// TwinCAT 3 PLC project step_motor
// ProgramVersion: 3.1.4023.0
// libraries:
//   Tc2_MC2, * (Beckhoff Automation GmbH)
//   Tc2_Standard, * (Beckhoff Automation GmbH)
//   Tc2_System, * (Beckhoff Automation GmbH)
//   Tc3_Module, * (Beckhoff Automation GmbH)
//   VisuSymbols,3.5.10.0,System
// project tree:
//   DUTs/ ST_MC_Status.TcDUT
//   / GlobalTextList.TcGTLO, PlcTask.TcTTO, Visualization Manager.TcVMO (not stored)
//   GVLs/ GVL.TcGVL
//   POUs/ MAIN.TcPOU
//   VISUs/ Visualization.TcVIS
// real-time tasks:
//   TASK PlcTask: cycle T#10ms, priority 20, ADS port 350
// motion (NC):
//   TASK NC-Task 1 SAF: cycle T#2ms, priority 4, ADS port 501
//   TASK NC-Task 1 SVB: cycle T#10ms, priority 8, ADS port 511
//   AXIS Axis 1 (id 1)
//     PositionAreaControl: Enable=false
//     TargetPosControl: Enable=false
//     OtherSettings: AllowMotionCmdToSlave=true
//     encoder EncType=4
//       EncPara: MaxCount=#x0000ffff
//         FilterTime: TPos=0.04, TVelo=0.1, TAcc=0.15
//         Inc: RefMode=2, RefSoftSyncMask=#x0000ffff
//     drive DrvType=24
//       Analog: VeloReferenz=800, TorqueSetpointScale=10, ScaleFactorActTorque=0.1
//       TimeComp: TaskDelayCycles=1
//     controller CtrType=1
//       CtrPara: PriorControlFactor=1
//         PosDiffControl: Enable=false
//         Observer: BandWidth=20
// I/O:
//   DEVICE Device 1 (EtherCAT), AmsNetId 5.59.220.46.2.1
//     Term 7 (EK1200) [EK1200-5000 EtherCAT Power supply (2A E-Bus)]
//       Term 8 (EL1008) [EL1008 8Ch. Dig. Input 24V, 3ms]
//       Term 9 (EL2008) [EL2008 8Ch. Dig. Output 24V, 0.5A]
//       Term 10 (EL3062) [EL3062 2Ch. Ana. Input 0-10V]
//       Term 11 (EL4002) [EL4002 2Ch. Ana. Output 0-10V, 12bit]
//       Term 12 (EL7031) [EL7031 1Ch. Stepper motor output stage (24V, 1.5A)]
//       Term 13 (EK1110) [EK1110 EtherCAT extension]
// variable links:
//   NC-Task 1 SAF/Axes/Axis 1 <-> Device 1 (EtherCAT)/Term 7 (EK1200)/Term 12 (EL7031)
//     Drive/Inputs/In/nState1 @bit 3 <-> STM Status/Status/Error
//     Drive/Inputs/In/nState1 @bit 5 <-> STM Status/Status/Moving negative
//     Drive/Inputs/In/nState1 @bit 4 <-> STM Status/Status/Moving positive
//     Drive/Inputs/In/nState1 @bit 1 <-> STM Status/Status/Ready
//     Drive/Inputs/In/nState1 <-> STM Status/Status/Ready to enable
//     Drive/Inputs/In/nState1 @bit 6 <-> STM Status/Status/Torque reduced
//     Drive/Inputs/In/nState1 @bit 2 <-> STM Status/Status/Warning
//     Drive/Inputs/In/nState2 @bit 3 <-> STM Status/Status/Digital input 1
//     Drive/Inputs/In/nState2 @bit 4 <-> STM Status/Status/Digital input 2
//     Drive/Inputs/In/nState2 @bit 5 <-> STM Status/Status/Sync error
//     Drive/Inputs/In/nState2 @bit 7 <-> STM Status/Status/TxPDO Toggle
//     Drive/Inputs/In/nState4 @bit 1 <-> WcState/InputToggle
//     Drive/Inputs/In/nState4 <-> WcState/WcState
//     Drive/Outputs/Out/nCtrl1 <-> STM Control/Control/Enable
//     Drive/Outputs/Out/nCtrl1 @bit 2 <-> STM Control/Control/Reduce torque
//     Drive/Outputs/Out/nCtrl1 @bit 1 <-> STM Control/Control/Reset
//     Drive/Outputs/Out/nDataOut2[0] <-> STM Velocity/Velocity
//     Enc/Inputs/In/nDataIn1[0] <-> ENC Status compact/Counter value
//     Enc/Inputs/In/nDataIn2[0] <-> ENC Status compact/Latch value
//     Enc/Inputs/In/nState1 @bit 4 <-> ENC Status compact/Status/Counter overflow
//     Enc/Inputs/In/nState1 @bit 3 <-> ENC Status compact/Status/Counter underflow
//     Enc/Inputs/In/nState1 @bit 1 <-> ENC Status compact/Status/Latch extern valid
//     Enc/Inputs/In/nState1 @bit 2 <-> ENC Status compact/Status/Set counter done
//     Enc/Inputs/In/nState2 @bit 4 <-> ENC Status compact/Status/Status of extern latch
//     Enc/Inputs/In/nState2 @bit 5 <-> ENC Status compact/Status/Sync error
//     Enc/Inputs/In/nState2 @bit 7 <-> ENC Status compact/Status/TxPDO Toggle
//     Enc/Inputs/In/nState4 @bit 1 <-> WcState/InputToggle
//     Enc/Inputs/In/nState4 <-> WcState/WcState
//     Enc/Outputs/Out/nCtrl1 @bit 3 <-> ENC Control compact/Control/Enable latch extern on negative edge
//     Enc/Outputs/Out/nCtrl1 @bit 1 <-> ENC Control compact/Control/Enable latch extern on positive edge
//     Enc/Outputs/Out/nCtrl1 @bit 2 <-> ENC Control compact/Control/Set counter
//     Enc/Outputs/Out/nDataOut1[0] <-> ENC Control compact/Set counter value
//   step_motor/step_motor Instance <-> NC-Task 1 SAF/Axes/Axis 1
//     PlcTask Inputs/MAIN.Axis.NcToPlc <-> Outputs/ToPlc
//     PlcTask Outputs/MAIN.Axis.PlcToNc <-> Inputs/FromPlc

CONFIGURATION step_motor
    RESOURCE PLC ON TwinCAT3
        TASK PlcTask(INTERVAL := T#10ms, PRIORITY := 20);
        PROGRAM MAIN WITH PlcTask : MAIN;
    END_RESOURCE
END_CONFIGURATION

// ---- DUTs/ST_MC_Status.TcDUT
TYPE ST_MC_Status :
STRUCT
	Status 		: BOOL;
	Done   		: BOOL;
	Busy   		: BOOL;
	Error  		: BOOL;
	Active 		: BOOL;
	CadAborted	: BOOL;
	InVelocity	: BOOL;
	ErrorID		: UDINT;
END_STRUCT
END_TYPE

// ---- GVLs/GVL.TcGVL
{attribute 'qualified_only'}
VAR_GLOBAL
	// Axis
	Axis: AXIS_REF;
	
	// Function blocks
	fbPowerAxis: MC_Power;
	fbMoveContinuous: MC_MoveContinuousRelative;
	
	// Parameters
	
	PowerOverride	: LREAL := 100;
	
	// Status
	
	Power 		  : ST_MC_Status;
	MoveRelative  : ST_MC_Status;
	Jog			  : ST_MC_Status;
END_VAR

// ---- POUs/MAIN.TcPOU
PROGRAM MAIN
VAR
	fbPowerAxis: MC_Power;
	fbMoveContinuous  : MC_MoveContinuousRelative;
	MC_Jog : MC_Jog;
		
	Axis: AXIS_REF;
	bExecute, bEnable: BOOL;
    bEnableP, bEnableN: BOOL := TRUE;
	rVelocity : LREAL := 600;
	rDistance : LREAL := 360;
END_VAR

GVL.fbPowerAxis(
	Axis:= GVL.Axis,
	Enable:= bEnable, 
	Enable_Positive:= bEnableP, 
	Enable_Negative:= bEnableN, 
	Override:= GVL.PowerOverride, 
	BufferMode:= MC_Aborting, 
	Options:= , 
	Status=> GVL.Power.Status, 
	Busy=> GVL.Power.Busy, 
	Active=> GVL.Power.Active, 
	Error=> GVL.Power.Error, 
	ErrorID=> gvl.Power.ErrorID);
	
	
(*GVL.fbMoveContinuous(
	Axis:= GVL.Axis, 
	Execute:= bExecute, 
	Distance:= rDistance, 
	Velocity:= rVelocity, 
	EndVelocity:= rVelocity, 
	Acceleration:= 500, 
	Deceleration:= 500, 
	Jerk:= 10, 
	BufferMode:= MC_Aborting, 
	Options:= , 
	InEndVelocity=> GVL.MoveRelative.InVelocity, 
	Busy=> GVL.MoveRelative.Busy, 
	Active=> GVL.MoveRelative.Active, 
	CommandAborted=> GVL.MoveRelative.CadAborted, 
	Error=> GVL.MoveRelative.Error, 
	ErrorID=> GVL.MoveRelative.ErrorID);*)
	
	(*MC_Jog(
	Axis:= GVL.Axis, 
	JogForward:= , 
	JogBackwards:= , 
	Mode:= MC_JOGMODE_CONTINOUS, 
	Position:= rDistance, 
	Velocity:= rVelocity, 
	Acceleration:= 500, 
	Deceleration:= 500, 
	Jerk:= 10, 
	Done=> GVL.Jog.Done, 
	Busy=> GVL.Jog.Busy, 
	Active=> GVL.Jog.Active, 
	CommandAborted=> GVL.Jog.CadAborted, 
	Error=> GVL.Jog.Error, 
	ErrorID=> GVL.Jog.ErrorID);*)

END_PROGRAM

// ---- GlobalTextList.TcGTLO
TEXTLIST GlobalTextList
  92 = 'enable mc_power'
  856 = 'execute mc_move'
  178 = 'velocity'
END_TEXTLIST

// ---- VISUs/Visualization.TcVIS
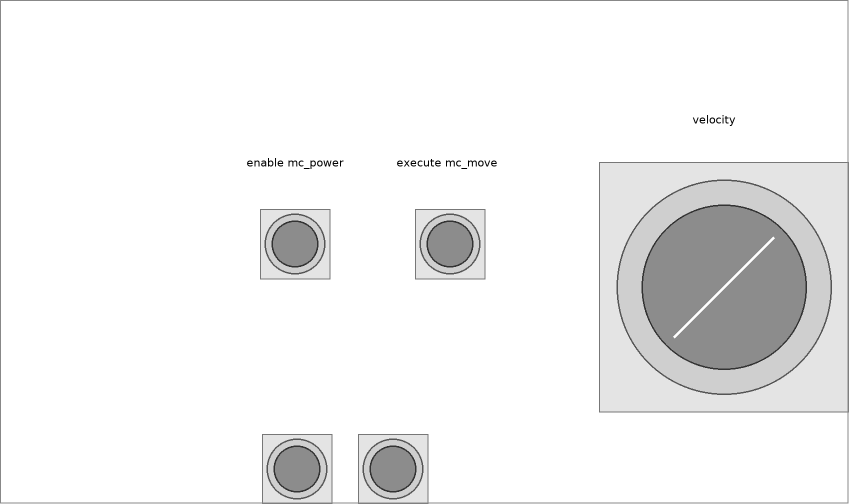
VISUALIZATION Visualization  // 849x504
    PushSwitchLed (260,209 70x70), variable: MAIN.bEnable, behaviour: TOGGLE, style: Switch-PushSwitchLed-Gray
    PushSwitchLed (415,209 70x70), variable: MAIN.bExecute, behaviour: TOGGLE, style: Switch-PushSwitchLed-Gray
    Label (220,148 150x30), "enable mc_power"
    Label (372,148 150x30), "execute mc_move"
    Potentiometer360 (599,162 250x250), variable: MAIN.rVelocity, style: Potentiometer-Potentiometer360-Gray, scale format: %.1f, scale 0..5000
        p2431819421: Outside
    Label (639,105 150x30), "velocity"
    PushSwitchLed (262,434 70x70), variable: MAIN.MC_Jog.JogForward, behaviour: TOGGLE, style: Switch-PushSwitchLed-Gray
    PushSwitchLed (358,434 70x70), variable: MAIN.MC_Jog.JogBackwards, behaviour: TOGGLE, style: Switch-PushSwitchLed-Gray
END_VISUALIZATION
